// Block: Areas_ITF

DATA_BLOCK Areas_ITF
VERSION : 0.1
   NON_RETAIN
   VAR
      A01 : ITF_A01;
      A02 : ITF_A02;
      A03 : ITF_A03;
      A04 : ITF_A04;
      AG : ITF_AG;
      Prod : ITF_ProductionMng;
   END_VAR

BEGIN
   // No initialization required
END_DATA_BLOCK
